{attribute 'linkalways'} 
{attribute 'no_explicit_call' := 'This FB is a CLASS and must be accessed using methods or properties'}
{attribute 'enable_dynamic_creation'}
FUNCTION_BLOCK FINAL MUL_SINT EXTENDS Node
VAR
	in1 : _SINT(0);
	in2 : _SINT(0);
	out : _SINT(0);
END_VAR

METHOD PUBLIC Clone : I_Node
VAR
	pNode : POINTER TO MUL_SINT;
END_VAR
pNode := __NEW(MUL_SINT);
Clone := pNode^;
END_METHOD

METHOD FB_init : BOOL
VAR_INPUT
	bInitRetains : BOOL; // if TRUE, the retain variables are initialized (warm start / cold start)
	bInCopyCode : BOOL;  // if TRUE, the instance afterwards gets moved into the copy code (online change)
END_VAR
AddInput('in1',THIS^.in1);
AddInput('in2',THIS^.in2);
AddOutput('out', THIS^.out);
END_METHOD

METHOD PROTECTED OnExecute
VAR
END_VAR
out.Value := in1.Value * in2.Value;
END_METHOD

END_FUNCTION_BLOCK

(* stored: Version 1.1.0.1, ProductVersion 3.1.4024.15
   POU MUL_SINT: Id {30f43430-5690-45e4-9080-5a66b5191a8e}, SpecialFunc None
   Folder Constructor: Id {674279b8-5c0f-4843-83a1-fd44e1831830}
   Method Clone: Id {a0aeebf0-3b8f-4e08-b9d1-a56194a3ca4f}
   Method FB_init: Id {4dad880c-4e38-49a4-ade0-28d206574e4b}
   Method OnExecute: Id {a855311a-ce76-4229-94c3-a13d022ae16a} *)
